{attribute 'TcGenerated'}
{attribute 'no-analysis'}
{attribute 'linkalways'}
// This function has been automatically generated from the project information.
VAR_GLOBAL CONSTANT
	{attribute 'const_non_replaced'}
	stLibVersion_BeckhoffHttpClient : ST_LibVersion := (iMajor := 1, iMinor := 1, iBuild := 0, iRevision := 0, nFlags := 0, sVersion := '1.1');
END_VAR

(* stored: Version 1.1.0.1, ProductVersion 3.1.4024.3
   GVL Global_Version: Id {4b2436a5-29d9-4dcb-a599-34dae6c9cf43} *)
